// TIA Portal V18 export
TYPE "UDT_sireneIO"
// stored: IsFailsafeCompliant false
   STRUCT
      O_sir_start { ExternalVisible := 'False'; ExternalWritable := 'False'} : Bool;
      O_sirena_1 { ExternalVisible := 'False'; ExternalWritable := 'False'} : Bool;
      O_sirena_2 { ExternalVisible := 'False'; ExternalWritable := 'False'} : Bool;
      O_sirena_3 { ExternalVisible := 'False'; ExternalWritable := 'False'} : Bool;
      O_sirena_4 { ExternalVisible := 'False'; ExternalWritable := 'False'} : Bool;
      O_sirena_5 { ExternalVisible := 'False'; ExternalWritable := 'False'} : Bool;
      O_sirena_6 { ExternalVisible := 'False'; ExternalWritable := 'False'} : Bool;
   END_STRUCT;
END_TYPE
